FUNCTION Convert_LWORD_TO_WORD : Hresult
VAR_INPUT
	in : LWORD;
	out : REFERENCE TO WORD;
END_VAR
VAR
	converted : WORD;
END_VAR

converted := LWORD_TO_WORD(in);

IF (WORD_TO_LWORD(converted) <> in) THEN
	Convert_LWORD_TO_WORD := INCOMPATIBLE;
	RETURN;
END_IF

out := converted;

END_FUNCTION

(* stored: Version 1.1.0.1, ProductVersion 3.1.4024.12
   POU Convert_LWORD_TO_WORD: Id {f7f159f1-ac3b-4b30-8b0e-6e47867785af}, SpecialFunc None *)
